{attribute 'GeneratedUsingTerminal: KL8610'}
{attribute addProperty BoxType "KL8610"}
{attribute addProperty Description ""}
{attribute addProperty Physics ""}
{attribute addProperty Id "KL8601_1AT %Q*KL_6576A6810"}
{attribute addProperty CRC "3312570472"}
{attribute addProperty Size "0"}
TYPE KL8610_C571D068 :
STRUCT
	{attribute addProperty Name "KL8601_1"}
	KL8601_1 : KL_6576A681;
END_STRUCT
END_TYPE

(* stored: Version 1.2.0.0, ProductVersion 3.1.4024.9
   DUT KL8610_C571D068: Id {ba3078a1-8332-426a-b347-cca5a0880881} *)
